(* CODESYS project elevator2.project

Project tree, tasks and I/O mapping:
  Device : CODESYS Control Win V3, 3S - Smart Software Solutions GmbH, version 3.5.12.10
    application Application
      libraries: Standard, * (System)
      task MainTask (cyclic, interval t#20ms, priority 1) calls PLC_PRG
      task VISU_TASK (cyclic, interval 100 ms, priority 31) calls VisuElems.Visu_Prg
      program PLC_PRG [ST]
      visualisation Visualization
  libraries: VisuSymbols, 3.5.10.0 (System)
  text list GlobalTextList
*)

// Device/Application/PLC_PRG
PROGRAM PLC_PRG
VAR
    // Inputs
    CallGround, CallFloor1, CallFloor2, CallFloor3: BOOL;
    FloorSensor0, FloorSensor1, FloorSensor2, FloorSensor3: BOOL;
    DoorClosed: BOOL;
    EmergencyStop: BOOL;

    // Outputs
    OpenDoor: BOOL := FALSE;
    CloseDoor: BOOL := FALSE;

    // Internal Variables
    TargetFloors: ARRAY[0..3] OF BOOL := [FALSE, FALSE, FALSE, FALSE];
    CurrentFloor: INT := 0;
    DoorTimer: TON;
    CloseDoorTimer: TON;
    MoveDelayTimer: TON;
    DoorOpen: BOOL := FALSE;
    MovingUp: BOOL := FALSE;
    MovingDown: BOOL := FALSE;
    i: INT;
	
	// Door Open-Close Animation
	aniDoor0, aniDoor1, aniDoor2, aniDoor3: DINT := 0;
END_VAR

// Determine Current Floor Based on Sensor Inputs
IF FloorSensor0 THEN CurrentFloor := 0; END_IF;
IF FloorSensor1 THEN CurrentFloor := 1; END_IF;
IF FloorSensor2 THEN CurrentFloor := 2; END_IF;
IF FloorSensor3 THEN CurrentFloor := 3; END_IF;

// Register Calls
IF CallGround THEN TargetFloors[0] := TRUE; END_IF;
IF CallFloor1 THEN TargetFloors[1] := TRUE; END_IF;
IF CallFloor2 THEN TargetFloors[2] := TRUE; END_IF;
IF CallFloor3 THEN TargetFloors[3] := TRUE; END_IF;

// Emergency Stop Handling
IF EmergencyStop THEN
    OpenDoor := FALSE;
    CloseDoor := FALSE;
    DoorOpen := FALSE;
    RETURN;
END_IF;

////////////////////////////////////////////////
// Lift Control Logic - Step-by-Step Movement //
////////////////////////////////////////////////

IF TargetFloors[CurrentFloor] THEN
    // Stop at requested floor
    CloseDoor := FALSE;
    TargetFloors[CurrentFloor] := FALSE; // Clear the request
    DoorTimer(IN := TRUE, PT := T#2S); // 2-second delay for door opening
    IF DoorTimer.Q THEN
        OpenDoor := TRUE;
        DoorOpen := TRUE;
    END_IF;
ELSIF DoorOpen THEN
    // Close door before moving
    OpenDoor := FALSE;
    CloseDoor := TRUE;
    DoorOpen := FALSE;
    CloseDoorTimer(IN := TRUE, PT := T#2S); // 2-second delay for door closing
ELSIF CloseDoorTimer.Q AND DoorClosed THEN
    // Determine next floor to move towards
    IF MovingUp THEN
        FOR i := CurrentFloor + 1 TO 3 DO
            IF TargetFloors[i] THEN
                // Request found, move up
                MoveDelayTimer(IN := TRUE, PT := T#500MS); // 500ms delay before moving
                IF MoveDelayTimer.Q THEN
                    MovingUp := TRUE;
                    MovingDown := FALSE; // Stop moving down if moving up *)
                    RETURN;
                END_IF;
            END_IF;
        END_FOR;

        // If no higher requests, move down
        IF NOT MovingDown THEN
            MovingUp := FALSE;
            MovingDown := TRUE;
        END_IF;
    END_IF;

    IF MovingDown THEN
        FOR i := CurrentFloor - 1 TO 0 BY -1 DO
            IF TargetFloors[i] THEN
                // Request found, move down
                MoveDelayTimer(IN := TRUE, PT := T#500MS); // 500ms delay before moving
                IF MoveDelayTimer.Q THEN
                    MovingDown := TRUE;
                    MovingUp := FALSE; // Stop moving up if moving down
                    RETURN;
                END_IF;
            END_IF;
        END_FOR;

        // If no lower requests, move up
        IF NOT MovingUp THEN
            MovingDown := FALSE;
            MovingUp := TRUE;
        END_IF;
    END_IF;
END_IF;

// Door Open-Close Animation

IF OpenDoor AND aniDoor0 < 70 AND CallGround THEN
    aniDoor0 := aniDoor0 + 1;
END_IF
IF CloseDoor AND aniDoor0 > 0 THEN
    aniDoor0 := aniDoor0 - 1;
END_IF

IF OpenDoor AND aniDoor1 < 70 AND CallFloor1 THEN
    aniDoor1 := aniDoor1 + 1;
END_IF
IF CloseDoor AND aniDoor1 > 0 THEN
    aniDoor1 := aniDoor1 - 1;
END_IF

IF OpenDoor AND aniDoor2 < 70 AND CallFloor2 THEN
    aniDoor2 := aniDoor2 + 1;
END_IF
IF CloseDoor AND aniDoor2 > 0 THEN
    aniDoor2 := aniDoor2 - 1;
END_IF

IF OpenDoor AND aniDoor3 < 70 AND CallFloor3 THEN
    aniDoor3 := aniDoor3 + 1;
END_IF
IF CloseDoor AND aniDoor3 > 0 THEN
    aniDoor3 := aniDoor3 - 1;
END_IF

// End Program...

END_PROGRAM

// Device/Application/Visualization
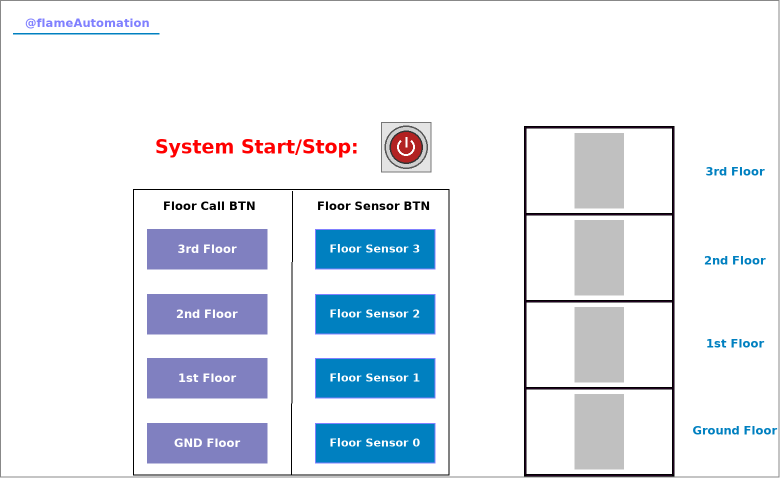
VISUALIZATION Visualization  // 780x478
    Group (133,189 316x286)
        Rectangle (0,0 316x286)
        Label (15,5 123x24), "Floor Call BTN"
        Rectangle (14,234 120x40), "GND Floor", colour toggle: PLC_PRG.CallGround
            toggle PLC_PRG.CallGround
        Rectangle (14,169 120x40), "1st Floor", colour toggle: PLC_PRG.CallFloor1
            toggle PLC_PRG.CallFloor1
        Rectangle (14,105 120x40), "2nd Floor", colour toggle: PLC_PRG.CallFloor2
            toggle PLC_PRG.CallFloor2
        Rectangle (14,40 120x40), "3rd Floor", colour toggle: PLC_PRG.CallFloor3
            toggle PLC_PRG.CallFloor3
        Rectangle (182,234 120x40), "Floor Sensor 0"
            toggle PLC_PRG.FloorSensor0
        Rectangle (182,169 120x40), "Floor Sensor 1"
            toggle PLC_PRG.FloorSensor1
        Rectangle (182,105 120x40), "Floor Sensor 2"
            toggle PLC_PRG.FloorSensor2
        Rectangle (182,40 120x40), "Floor Sensor 3"
            toggle PLC_PRG.FloorSensor3
        Label (179,5 123x24), "Floor Sensor BTN"
        Line (159,2) (158,285)
    Group (489,131 220x340)
        Group (0,261 220x79)
            Rectangle (88,2 45x75)
            Rectangle (73,2 40x75)
                p3560616238: PLC_PRG.aniDoor0
            Rectangle (108,2 40x75)
                p3560616238: -PLC_PRG.aniDoor0
            Rectangle (0,0 85x79)
            Rectangle (135,0 85x79)
        Group (0,174 220x79)
            Rectangle (88,2 45x75)
            Rectangle (73,2 40x75)
                p3560616238: PLC_PRG.aniDoor1
            Rectangle (108,2 40x75)
                p3560616238: -PLC_PRG.aniDoor1
            Rectangle (0,0 85x79)
            Rectangle (135,0 85x79)
        Group (0,87 220x79)
            Rectangle (88,2 45x75)
            Rectangle (73,2 40x75)
                p3560616238: PLC_PRG.aniDoor2
            Rectangle (108,2 40x75)
                p3560616238: -PLC_PRG.aniDoor2
            Rectangle (0,0 85x79)
            Rectangle (135,0 85x79)
        Group (0,0 220x79)
            Rectangle (88,2 45x75)
            Rectangle (73,2 40x75)
                p3560616238: PLC_PRG.aniDoor3
            Rectangle (108,2 40x75)
                p3560616238: -PLC_PRG.aniDoor3
            Rectangle (0,0 85x79)
            Rectangle (135,0 85x79)
    Group (524,126 150x350)
        Rectangle (0,87 150x2)
        Rectangle (0,174 150x2)
        Rectangle (0,261 150x2)
        Rectangle (0,348 150x2)
        Rectangle (0,0 150x2)
        Rectangle (148,0 2x349)
        Rectangle (0,0 2x349)
    Group (692,153 86x296)
        Label (0,259 86x37), "Ground Floor"
        Label (0,172 86x37), "1st Floor"
        Label (0,89 86x37), "2nd Floor"
        Label (0,0 86x37), "3rd Floor"
    Label (26,11 123x24), "@flameAutomation"
    Rectangle (13,33 146x1)
    Group (143,122 288x50)
        PowerSwitch (238,0 50x50), variable: PLC_PRG.EmergencyStop, behaviour: TAP, style: Switch-PowerSwitch-Red
        Label (0,13 228x24), "System Start/Stop:"
END_VISUALIZATION
